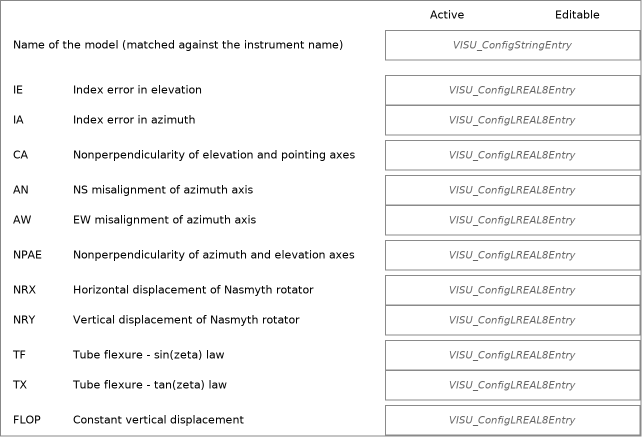
VISUALIZATION VISU_AxesPointingModelConfig_part1  // 642x437
VAR_IN_OUT
    active : AxesPointingModelConfig;
    editable : AxesPointingModelConfig;
END_VAR
    Label (385,5 125x20), "Active"
    Label (515,5 125x20), "Editable"
    Label (10,75 30x30), "IE"
    Frame (385,75 255x30)
        shows VISU_ConfigLREAL8Entry(active := active.IE, editable := editable.IE)
    Label (70,75 315x30), "Index error in elevation"
    Label (10,105 30x30), "IA"
    Frame (385,105 255x30)
        shows VISU_ConfigLREAL8Entry(active := active.IA, editable := editable.IA)
    Label (70,105 315x30), "Index error in azimuth"
    Label (10,140 30x30), "CA"
    Frame (385,140 255x30)
        shows VISU_ConfigLREAL8Entry(active := active.CA, editable := editable.CA)
    Label (70,140 315x30), "Nonperpendicularity of elevation and pointing axes"
    Label (10,175 30x30), "AN"
    Frame (385,175 255x30)
        shows VISU_ConfigLREAL8Entry(active := active.AN, editable := editable.AN)
    Label (70,175 315x30), "NS misalignment of azimuth axis"
    Frame (385,205 255x30)
        shows VISU_ConfigLREAL8Entry(active := active.AW, editable := editable.AW)
    Label (10,205 60x30), "AW"
    Label (70,205 315x30), "EW misalignment of azimuth axis"
    Frame (385,240 255x30)
        shows VISU_ConfigLREAL8Entry(active := active.NPAE, editable := editable.NPAE)
    Label (10,240 60x30), "NPAE"
    Label (70,240 315x30), "Nonperpendicularity of azimuth and elevation axes"
    Frame (385,275 255x30)
        shows VISU_ConfigLREAL8Entry(active := active.NRX, editable := editable.NRX)
    Label (10,275 60x30), "NRX"
    Label (70,275 315x30), "Horizontal displacement of Nasmyth rotator"
    Frame (385,305 255x30)
        shows VISU_ConfigLREAL8Entry(active := active.NRY, editable := editable.NRY)
    Label (10,305 60x30), "NRY"
    Label (70,305 315x30), "Vertical displacement of Nasmyth rotator"
    Frame (385,340 255x30)
        shows VISU_ConfigLREAL8Entry(active := active.TF, editable := editable.TF)
    Label (10,340 60x30), "TF"
    Label (70,340 315x30), "Tube flexure - sin(zeta) law"
    Frame (385,370 255x30)
        shows VISU_ConfigLREAL8Entry(active := active.TX, editable := editable.TX)
    Label (10,370 60x30), "TX"
    Label (70,370 315x30), "Tube flexure - tan(zeta) law"
    Frame (385,30 255x30)
        shows VISU_ConfigStringEntry(active := active.name, editable := editable.name)
    Label (10,30 370x30), "Name of the model (matched against the instrument name)"
    Frame (385,405 255x30)
        shows VISU_ConfigLREAL8Entry(active := active.FLOP, editable := editable.FLOP)
    Label (10,405 60x30), "FLOP"
    Label (70,405 315x30), "Constant vertical displacement"
END_VISUALIZATION

(* stored: Version 1.1.0.1, ProductVersion 3.1.4019.2
   Visu VISU_AxesPointingModelConfig_part1: Id {5ca43030-9abc-4c82-9f21-f71c013a4d41} *)
